// TwinCAT 3 PLC project MasterPLC
// ProgramVersion: 3.1.4024.0
// libraries:
//   Tc2_Standard, * (Beckhoff Automation GmbH)
//   Tc2_System, * (Beckhoff Automation GmbH)
//   Tc3_Module, * (Beckhoff Automation GmbH)
// project tree:
//   / PlcTask.TcTTO
//   POUs/ MAIN.TcPOU
// real-time tasks:
//   TASK PlcTask: cycle T#10ms, priority 20, ADS port 350
// motion (NC):
//   TASK NC-Task 1 SAF: cycle T#2ms, priority 4, ADS port 501
//   TASK NC-Task 1 SVB: cycle T#10ms, priority 8, ADS port 511
//   AXIS Axis 1 (id 1)
//     OtherSettings: AllowMotionCmdToSlave=true
//     encoder EncType=19
//       EncPara: MaxCount=#xffffffff
//     drive DrvType=16
//       DrvPara: MaxCount=#xffffffff, DriveControlDWord=#x00000100
//         Analog: TorqueSetpointScale=10, ScaleFactorActTorque=0.1
//         TimeComp: TaskDelayCycles=1
//     controller CtrType=1
//       CtrPara: PriorControlFactor=1
//         Observer: BandWidth=20
// I/O:
//   DEVICE Device 3 (EtherCAT), AmsNetId 5.78.205.182.4.1
//     Drive 1 (SB4-C680) [SB4-C680]
// variable links:
//   NC-Task 1 SAF/Axes/Axis 1 <-> Device 3 (EtherCAT)/Drive 1 (SB4-C680)
//     Drive/Inputs/In/nDataIn1 <-> TxPdoMapping1/Following error actual value
//     Drive/Inputs/In/nState1 <-> TxPdoMapping1/Statusword
//     Drive/Inputs/In/nState2 <-> TxPdoMapping1/Statusword @bit 8
//     Drive/Inputs/In/nState4 @bit 1 <-> WcState/InputToggle
//     Drive/Inputs/In/nState4 <-> WcState/WcState
//     Drive/Inputs/In/nState5 <-> TxPdoMapping1/Modes of operation display
//     Drive/Outputs/Out/nCtrl1 <-> RxPdoMapping1/Controlword
//     Drive/Outputs/Out/nCtrl2 <-> RxPdoMapping1/Controlword @bit 8
//     Drive/Outputs/Out/nCtrl5 <-> RxPdoMapping1/Modes of operation
//     Drive/Outputs/Out/nDataOut1 <-> RxPdoMapping1/Target position
//     Drive/Outputs/Out/nDataOut2 <-> RxPdoMapping1/Target velocity
//     Enc/Inputs/In/nDataIn1 <-> TxPdoMapping1/Position actual value
//     Enc/Inputs/In/nDataIn7 <-> TxPdoMapping1/Velocity Actual Value
//     Enc/Inputs/In/nState4 @bit 1 <-> WcState/InputToggle
//     Enc/Inputs/In/nState4 <-> WcState/WcState

CONFIGURATION MasterPLC
    RESOURCE PLC ON TwinCAT3
        TASK PlcTask(INTERVAL := T#10ms, PRIORITY := 20);
        PROGRAM MAIN WITH PlcTask : MAIN;
    END_RESOURCE
END_CONFIGURATION

// ---- POUs/MAIN.TcPOU
PROGRAM MAIN
VAR
END_VAR

END_PROGRAM
